// TIA Portal V18 export
// export: Created 2026-03-12T16:04:34.4994018Z, ExportSetting WithDefaults, DisplayName Totally Integrated Automation Portal, DisplayVersion V18 Update 5, DisplayName TIA Portal Openness, DisplayVersion V18 Update 5, DisplayName TIA Portal Version Control Interface, DisplayVersion V18, DisplayName SINAMICS Startdrive Advanced, DisplayVersion V18, DisplayName SINAMICS Startdrive G130, G150, S120, S150, SINAMICS MV, S210, DisplayVersion V18, DisplayName SINAMICS Startdrive G110M, G120, G120C, G120D, G120P, G115D, DisplayVersion V18, DisplayName STEP 7 Professional, DisplayVersion V18 Update 5, DisplayName STEP 7 Safety, DisplayVersion V18, DisplayName WinCC Professional, DisplayVersion V18 Update 5
FUNCTION_BLOCK "FB_PARTIDA_INVERSOR"   // FB11, LAD
TITLE = Function Block PARTIDA INVERSOR
{ S7_Optimized_Access := 'TRUE' }
VERSION : 0.1
// Bloco para configurar os sinais de pulso (liga e desliga) em conjunto com 2 relés
// stored: AutoNumber true, IsIECCheckEnabled false, IsRetainMemResEnabled false, MemoryReserve 100, SetENOAutomatically false, UDAEnableTagReadback false
   VAR_INPUT
      IN_LIGA_BOMBA : Bool;   // Entrada do comando para ligar a bomba
      IN_SUCÇÃO_OK : Bool;   // 0 = Sucção OK, permite ligar a bomba
      IN_OBSTRUÇÃO : Bool;   // 0 = Obstrução na pista
      IN_SOBRETORQUE : Bool;   // 0 = Sobretorque do motor/bomba
      IN_FALHA : Bool;   // 1 = Bomba em falha, comando desliga é pulsado
      IN_LIGADO : Bool;   // 1 = Bomba Ligada
      IN_HABILITA_CMB : Bool;   // Habilita bomba (Principal / Reserva)
      IN_LIGA_BOMBA_AUTO : Bool;
   END_VAR
   VAR_OUTPUT
      OUT_LIGA : Bool;   // Saída digital para ligar o Inversor
      OUT_DESLIGA : Bool;   // Saída digital para desligar o Inversor
   END_VAR
   VAR
      TEMP_LIGA : IEC_TIMER;   // Temporizador para simular o pulso de liga (0.5s)
      TEMP_DESLIGA : IEC_TIMER;   // Temporizador para simular o pulso de desliga (0.5s)
      DESLIGA_BOMBA { S7_SetPoint := 'True'} : Bool;   // Memória auxiliar para desligar o Inversor
      OUT_TEST : Bool;
   END_VAR
BEGIN

REGION Network 1: Saída digital para ligar o Inversor
   // Condições para ligar:
   // IN_LIGA_BOMBA = 1, Sinal de liga recebido do bloco CONDIÇÃO DE PARTIDA
   // IN_SUCÇÃO = 1, Significa que a bomba está com sucção OK
   // IN_OBSTRUÇÃO = 0, Significa que não há obstrução na pista
   // IN_SOBRETORQUE = 0, Significa que não há alarme de sobretorque do motor/bomba
   // OUT_DESLIGA = 1, Para ligar, é necessário que a entrada digital de desliga no inversor (STOP) esteja com sinal alto, 
   // aguardando que o mesmo seja cortado com um pulso para desligar.
   // - Para desligar é necessário que o motor/bomba esteja enviando sinal de ligado.
   // 
   // Pulso para ligar: Configurado com um tempo de 0.5S
   // Pulso para desligar: Configurado com um tempo de 0.5S
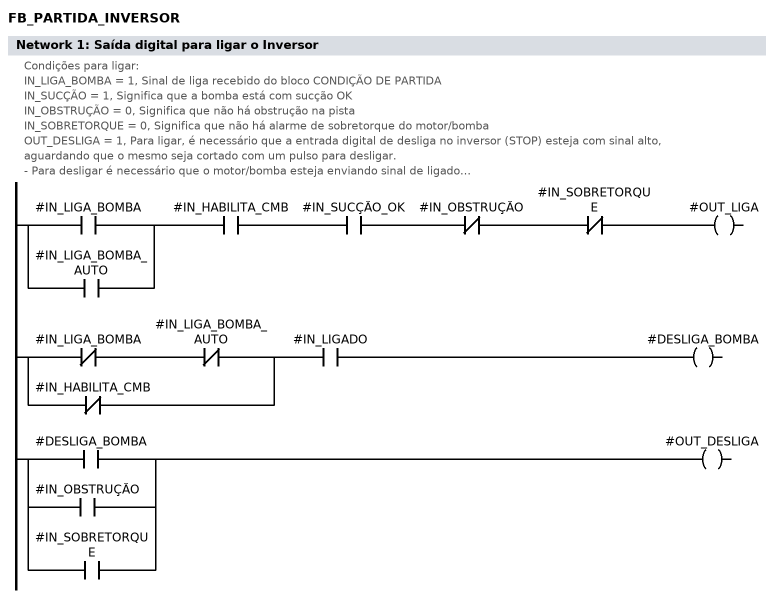
   RUNG wire#powerrail
      Contact( #IN_LIGA_BOMBA )
      wire#w1
      Contact( #IN_HABILITA_CMB )
      Contact( #IN_SUCÇÃO_OK )
      I_Contact( #IN_OBSTRUÇÃO )
      I_Contact( #IN_SOBRETORQUE )
      Coil( #OUT_LIGA )
   END_RUNG
   RUNG wire#powerrail
      Contact( #IN_LIGA_BOMBA_AUTO )
   END_RUNG wire#w1
   RUNG wire#powerrail
      I_Contact( #IN_LIGA_BOMBA )
      I_Contact( #IN_LIGA_BOMBA_AUTO )
      wire#w2
      Contact( #IN_LIGADO )
      Coil( #DESLIGA_BOMBA )
   END_RUNG
   RUNG wire#powerrail
      I_Contact( #IN_HABILITA_CMB )
   END_RUNG wire#w2
   RUNG wire#powerrail
      Contact( #DESLIGA_BOMBA )
      wire#w3
      Coil( #OUT_DESLIGA )
   END_RUNG
   RUNG wire#powerrail
      Contact( #IN_OBSTRUÇÃO )
   END_RUNG wire#w3
   RUNG wire#powerrail
      Contact( #IN_SOBRETORQUE )
   END_RUNG wire#w3
   // the same network as SCL:
   #OUT_LIGA := (#IN_LIGA_BOMBA OR #IN_LIGA_BOMBA_AUTO) AND #IN_HABILITA_CMB AND #IN_SUCÇÃO_OK AND NOT #IN_OBSTRUÇÃO AND NOT #IN_SOBRETORQUE;
   #DESLIGA_BOMBA := ((NOT #IN_LIGA_BOMBA AND NOT #IN_LIGA_BOMBA_AUTO) OR NOT #IN_HABILITA_CMB) AND #IN_LIGADO;
   #OUT_DESLIGA := #DESLIGA_BOMBA OR #IN_OBSTRUÇÃO OR #IN_SOBRETORQUE;
END_REGION
END_FUNCTION_BLOCK
